(* IEC 61131-3 sources: Industry-PLC-LLM/data/PLCBEAD_repo/PLCBEAD_PLCEmbed-main/PLC-BEAD/Source/GEB/TIMECHECK, 1 file *)

(* ---- TIMECHECK.ST ---- *)
FUNCTION TIMECHECK:BOOL

	VAR_INPUT
		TD :	UDINT;
		START :	UDINT;
		STOP :	UDINT;
	END_VAR

	IF STOP < START THEN
		TIMECHECK := START <= TD OR  TD < STOP;
	ELSE
		TIMECHECK := START <= TD AND TD < STOP;
	END_IF;

END_FUNCTION

PROGRAM program0
  VAR
	TD :	UDINT;
	START :	UDINT;
	STOP :	UDINT;
    CEIL5_OUT : BOOL;
  END_VAR

  CEIL5_OUT := TIMECHECK(TD, START, STOP);
END_PROGRAM
